SUBAPPLICATION Uebung_015b (* Object Pointer umschalten -- 3-fach *)
  (* Standard: 61499-2; Description: Copyright (c) 2026 Meisterschulen am Ostbahnhof This program and the accompanying materials are made available under the terms of the Eclipse Public License 2.0 which is available at https://www.eclipse.org/legal/epl-2.0/ SPDX-License-Identifier: EPL-2.0 *)
  (* Version 1.0, 2026-09-10, Franz Höpfinger, Meisterschulen am Ostbahnhof, initial API and implementation and/or initial documentation *)
  PACKAGE Uebungen;
  IMPORT isobus::UT::io::Softkey::SoftKeyActivationCode::SK_RELEASED;
  IMPORT Uebungen::const::UT::DefaultPool::Button_A1;
  IMPORT Uebungen::const::UT::DefaultPool::Button_A2;
  IMPORT Uebungen::const::UT::DefaultPool::ObjectPointer_P1;
  IMPORT Uebungen::const::UT::DefaultPool::SoftKey_F1;
  IMPORT Uebungen::const::UT::DefaultPool::SoftKey_F2;
  IMPORT Uebungen::const::UT::DefaultPool::SoftKey_F3;
  IMPORT isobus::UT::Q::const::IDs::ID_NULL;
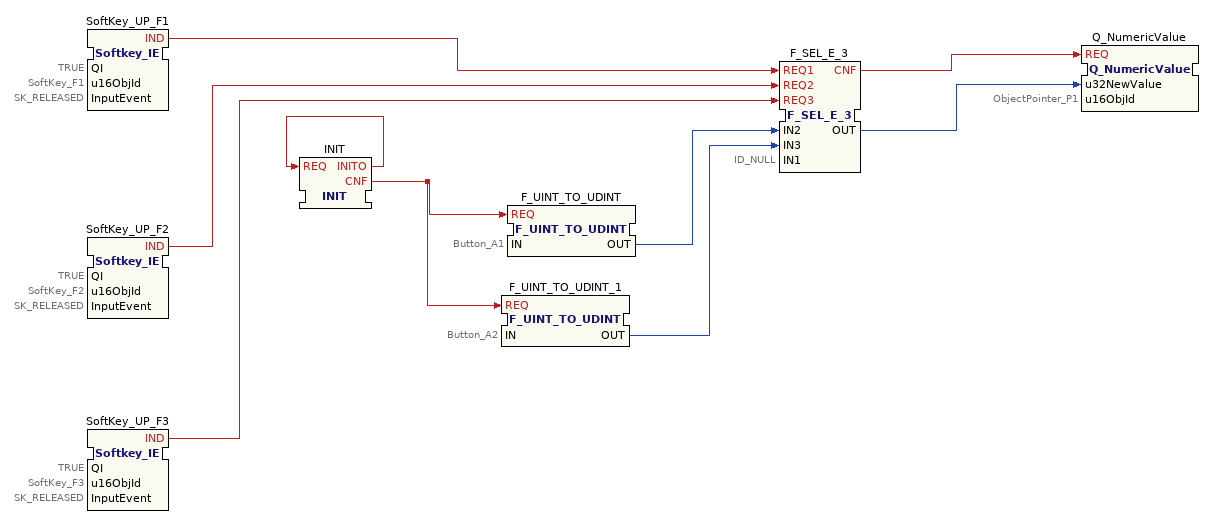
  FBS
    SoftKey_UP_F1 : isobus::UT::io::Softkey::Softkey_IE(QI := TRUE, u16ObjId := SoftKey_F1, InputEvent := SK_RELEASED);
    SoftKey_UP_F2 : isobus::UT::io::Softkey::Softkey_IE(QI := TRUE, u16ObjId := SoftKey_F2, InputEvent := SK_RELEASED);
    F_UINT_TO_UDINT : iec61131::conversion::F_UINT_TO_UDINT(IN := Button_A1);
    F_SEL_E_3 : eclipse4diac::utils::selection::F_SEL_E_3(IN1 := ID_NULL);
    Q_NumericValue : isobus::UT::Q::Q_NumericValue(u16ObjId := ObjectPointer_P1);
    SoftKey_UP_F3 : isobus::UT::io::Softkey::Softkey_IE(QI := TRUE, u16ObjId := SoftKey_F3, InputEvent := SK_RELEASED);
    F_UINT_TO_UDINT_1 : iec61131::conversion::F_UINT_TO_UDINT(IN := Button_A2);
    INIT : iec61131::booleanOperators::INIT;
  END_FBS
  EVENT_CONNECTIONS
    F_SEL_E_3.CNF TO Q_NumericValue.REQ;
    SoftKey_UP_F1.IND TO F_SEL_E_3.REQ1;
    SoftKey_UP_F2.IND TO F_SEL_E_3.REQ2;
    SoftKey_UP_F3.IND TO F_SEL_E_3.REQ3;
    INIT.INITO TO INIT.REQ;
    INIT.CNF TO F_UINT_TO_UDINT.REQ;
    INIT.CNF TO F_UINT_TO_UDINT_1.REQ;
  END_CONNECTIONS
  DATA_CONNECTIONS
    F_UINT_TO_UDINT.OUT TO F_SEL_E_3.IN2;
    F_SEL_E_3.OUT TO Q_NumericValue.u32NewValue;
    F_UINT_TO_UDINT_1.OUT TO F_SEL_E_3.IN3;
  END_CONNECTIONS
END_SUBAPPLICATION
